PROGRAM IO
VAR
END_VAR


LightBulb.StartSwitch 	:=	LightBulb.StartSignal;
LightBulb.StopSwitch	:=	LightBulb.StopSignal;

END_PROGRAM

(* stored: Version 1.1.0.1, ProductVersion 3.1.4024.9
   POU IO: Id {bf9a2bcf-91a0-40a3-a6e9-abaa1c5e0bea}, SpecialFunc None *)
